TYPE ST_CartInputDataPool :
STRUCT
	// cart information, import from other task
	m_cartStatus AT %I*:ST_CartStatus;
	
	// safety information, import from safety check task
	m_safetyData AT %I*: ST_SafetyData;
	
	// slave status, import from slave control task
	m_slaveStatus AT %I*: ST_SlaveStatus;
	
	//UI information, import from UI controller
	m_UIData :ST_CartUIData;
	
	
END_STRUCT
END_TYPE

(* stored: Version 1.1.0.1, ProductVersion 3.1.4024.11
   DUT ST_CartInputDataPool: Id {52655851-7a50-4c98-9a1e-ea6f4c6758df} *)
